// TIA Portal V19 export
DATA_BLOCK "ItemInfoScada"   // DB11
{ S7_Optimized_Access := 'TRUE' }
AUTHOR : FLA
FAMILY : UHT
VERSION : 1.0
// stored: AutoNumber false, MemoryReserve 0
   VAR
      Items : Array[1..85] of "ItemInfo_UDT";
   END_VAR
BEGIN
   // Items[1] : Y0101
   // Items[2] : Y0103
   // Items[3] : Y0104
   // Items[4] : Y0109
   // Items[5] : Y0111
   // Items[6] : Y0112
   // Items[7] : Y0113
   // Items[8] : Y0114
   // Items[9] : Y0115
   // Items[10] : M0139
   // Items[11] : Y0116
   // Items[12] : Y0108
   // Items[13] : Y0117
   // Items[14] : Y0118
   // Items[15] : Y0237
   // Items[16] : Y0238
   // Items[17] : Y0119
   // Items[18] : Y0124
   // Items[19] : Y0135_NOT_USED
   // Items[20] : Y0136_NOT_USED
   // Items[21] : Y0137_NOT_USED
   // Items[22] : Y0143
   // Items[23] : Y0144_NOT_USED
   // Items[24] : Y0147
   // Items[25] : Y0148
   // Items[26] : Y0158
   // Items[27] : Y0545
   // Items[28] : PACK1
   // Items[29] : PACK2
   // Items[30] : PACK3
   // Items[31] : PACK4
   // Items[32] : AlarmLamp
   // Items[33] : AHV_CLOSED
   // Items[34] : AHV_HIGH_LEVEL
   // Items[35] : AHV_READY
   // Items[36] : AHV_SHUT_DOWN
   // Items[37] : AHV_STERILE
   // Items[38] : PROD_AVAILABLE
   // Items[39] : RINSE_READY
   // Items[40] : CAUSTIC_READY
   // Items[41] : ACID_READY
   // Items[42] : CIP_FILLER_ENABLE
   // Items[43] : WATER_PUMP
   // Items[44] : Y0901
   // Items[45] : Y0902
   // Items[46] : Y0903
   // Items[47] : TANK_READY
   // Items[48] : TANK_OPEN
   // Items[49] : Y0904
   // Items[50] : Y0905
   // Items[51] : Y0906
   // Items[52] : Y0907
   // Items[53] : Y0908
   // Items[54] : Y0909
   // Items[55] : Y0910
   // Items[56] : Y0911
   // Items[57] : Y0912
   // Items[58] : Q41_1
   // Items[59] : CIP_Route
   // Items[60] : SIP_Steam
   // Items[61] : Product_Available
   // Items[62] : Barrier_Sterile
   // Items[63] : Product_Route
   // Items[64] : X0913
   // Items[65] : V0930
   // Items[66] : V0931
   // Items[67] : spare2
   // Items[68] : V0552
   // Items[69] : V0934
   // Items[70] : V0935
   // Items[71] : V0940
   // Items[72] : V0941
   // Items[73] : V0942
   // Items[74] : V0943
   // Items[75] : V0944
   // Items[76] : V0945
   // Items[77] : M0940
   // Items[78] : V1021
   // Items[79] : V1023
   // Items[80] : V1024
   // Items[81] : V1025
   // Items[82] : V1027
   // Items[83] : V1083
   // Items[84] : M0941
   // Items[85] : V0936
END_DATA_BLOCK
